// TIA Portal V20 export
DATA_BLOCK "WEBMON"   // DB43
{ S7_Optimized_Access := 'FALSE' }
VERSION : 0.1
// 표준 접근 : 외부 S7 통신(gr-console) 읽기용, 레이아웃은 LayoutSig 로 검증
// stored: AutoNumber true, DBAccessibleFromOPCUA true, DBAccessibleFromWebserver true, IsOnlyStoredInLoadMemory false, IsWriteProtectedInAS false
   VAR
      LayoutSig : DWord := 16#6FBC_9493;   // 레이아웃 서명 (gr-contract gen-sig 가 생성, 수동 수정 금지)
      UpdateTime : DTL;   // 갱신 시각 (PLC 로컬)
      Mode : Word;   // "MACHINE".Mode (MODE_* : 0 Boot, 1 Init, 2 Maint, 4 Standby, 8 Manual, 16 Ready, 32 Auto, 128 Fault, 256 Teach)
      Stat { S7_SetPoint := 'True'} : "LGR_Interface_GR_Status";   // "OPCUA".STAT 복사 (모드 / 상태 / StatusCode / Task Now·Queue·Completed·Canceled·Rejected / 측정 / 인터록 / 신호 / 드라이브)
      Proc { S7_SetPoint := 'True'} : "LGR_Proc_component";   // "TASK".Proc (진행 스텝 / 경과 시간 / 메시지)
      Alarm : Struct   // "MACHINE".Alarm 최근 코드
         Fault : Bool;
         Warn : Bool;
         FaultCode : Array[0..9] of UDInt;
         WarnCode : Array[0..9] of UDInt;
         EventCode : Array[0..9] of UDInt;
         TaskCode : Array[0..9] of UDInt;
      END_STRUCT;
      Axis : Array["X".."G"] of Struct   // "DRIVE".Axis 요약 (X, Y, Z, G)
         Position : Real;   // PV.Position (mm)
         Target : Real;   // SV.Position (mm)
         Speed : Real;
         Torque : Real;   // % mot
         LagError : Real;
         Ready : Bool;
         Enabled : Bool;
         Running : Bool;
         StandStill : Bool;
         MainCode : UInt;
         SubCode : UInt;
      END_STRUCT;
      Gripper : Struct
         ItemDetect : Bool;
         GID : Array[0..3] of Real;   // 레이저 거리 (L, F, R, B)
         FLD : Real;   // 바닥 거리
         TorqueReachedPosition : Real;
         State { S7_SetPoint := 'True'} : "LGR_GripperState";   // "MACHINE".Gripper.State (그리퍼 종합 상태 : TorqueReached / TorqueStop / Stall / StallTime …)
         Code : USInt;   // "GRIP".Status.Code (GRIP_ST_*)
         Timeout : USInt;   // "GRIP".Status.Timeout (GRIP_TO_*)
         Mode : USInt;   // "GRIP".Mode 진행 중 모드
         "Step" : Int;   // "GRIP".Step
         ErrorCode : Int;   // "GRIP".Result.ErrorCode (GRIP_E_*)
         Inch : Int;   // "GRIP".Result.Inch
         Busy : Bool;
         Done : Bool;
         Error : Bool;
         GripOk : Bool;
         ItemPresent : Bool;
         Obstacle : Bool;
         Thermal : Bool;
         AtSpeed : Bool;
         Contact : Bool;
         LimitNow : Real;   // 지금 보내는 토크 제한 (%)
         Mech : Real;   // 기구 부하 (%)
         Rise : Real;   // |PV.Torque| − Mech (%)
         TorqPct : Real;   // 적용 토크 (%)
         Force_N : Real;   // 타이어 힘 환산 (N)
         ContactPos : Real;
         ReachedPos : Real;
      END_STRUCT;
      Measure : Struct   // "FUNC" 측정 진행 상태
         Item : Struct
            Busy : Bool;
            Done : Bool;
            Reported : Bool;
            WorkCell : UInt;
            Code : UDInt;
            Status : UInt;
            InnerDia : Real;
            OffsetX : Real;
            OffsetY : Real;
            UpperBeadHeight : Real;
            TireHeight : Real;
            Torq_InnerDia : Real;
            InBusy : Bool;
            InDone : Bool;
            InValid : Bool;
            InInnerDia : Real;
            OutBusy : Bool;
            OutDone : Bool;
            OutValid : Bool;
            OutInnerDia : Real;
         END_STRUCT;
         Sku : Struct
            Enable : Bool;
            Busy : Bool;
            Done : Bool;
            WorkCell : UInt;
            StackCount : USInt;
            StackHeight : Real;
            EachHeight : Real;
            BeadPos : Array[0..19] of Real;
         END_STRUCT;
         Floor : Struct
            Enable : Bool;
            Busy : Bool;
            Done : Bool;
            Height : Real;
         END_STRUCT;
         LastBead : Struct
            Enable : Bool;
            Busy : Bool;
            Done : Bool;
            LastBeadPos : Real;
            PickZTarget : Real;
         END_STRUCT;
      END_STRUCT;
      MeasLog : Struct   // "MEASLOG" 요약
         Total : UDInt;
         Count : Int;
      END_STRUCT;
   END_VAR
BEGIN
END_DATA_BLOCK
